{attribute 'TcGenerated'}
{attribute 'no-analysis'}
{attribute 'linkalways'}
// This function has been automatically generated from the project information.
VAR_GLOBAL CONSTANT
	{attribute 'const_non_replaced'}
	stLibVersion_TcHAL : ST_LibVersion := (iMajor := 0, iMinor := 1, iBuild := 3, iRevision := 0, nFlags := 0, sVersion := '0.1.3');
END_VAR

(* stored: Version 1.1.0.1, ProductVersion 3.1.4024.6
   GVL Global_Version: Id {11f2dfac-c5ed-49c1-b978-d1062915f763} *)
